FUNCTION F_AND_REF : BOOL
VAR_IN_OUT
	bValueRoot		: BOOL;
END_VAR
VAR_INPUT
	bValueCombine	: BOOL;
END_VAR

bValueRoot := bValueRoot AND bValueCombine;

END_FUNCTION

(* stored: Version 1.1.0.1, ProductVersion 3.1.4024.11
   POU F_AND_REF: Id {c76f6170-b64e-4b2f-b2de-f02f911298d1}, SpecialFunc None *)
